{library PUBLIC}
TYPE GANTRY_ASYNC_FUNCTION_NUMBER :(

(* GoTo functions - No parameters *)
	GANTRY_ASYNC_FUNCTION_GOTO_HOME:=		11,
	GANTRY_ASYNC_FUNCTION_GOTO_STATION:=	12,

(* Pick Leav function
	ParameterW=Station 1-4*10 + position 1-9 + Station 1-4*1000 +position 1-9 * 100
 *)
	GANTRY_ASYNC_FUNCTION_PL:=					22			(* Pick/leave at position *)
);
END_TYPE

(* stored: Version 1.1.0.1, ProductVersion 3.1.4024.2
   EnumerationTextList GANTRY_ASYNC_FUNCTION_NUMBER: Id {fb504019-e7b4-442a-b60d-d049e506107f} *)
